FUNCTION_BLOCK FB_Device
VAR_INPUT
	inpAutomatic		: BOOL;
	inpSim				: BOOL := TRUE;
	
	cmdReset			: BOOL;
END_VAR
VAR_OUTPUT
END_VAR
VAR
END_VAR

PROPERTY ModeAutomatic : BOOL
GET
ModeAutomatic := inpAutomatic;
END_GET
END_PROPERTY

PROPERTY ModeManual : BOOL
GET
ModeManual := NOT inpAutomatic;
END_GET
END_PROPERTY

END_FUNCTION_BLOCK

(* stored: Version 1.1.0.1, ProductVersion 3.1.4024.4
   POU FB_Device: Id {df461c38-08f6-480c-a85c-0958733e653b}, SpecialFunc None
   Property ModeAutomatic: Id {15d02fd8-4ac5-4c34-9335-fe3f05621b5c}
   Get Get: Id {1cf7cdfc-1822-48eb-8dea-c7f604a7f1ff}
   Property ModeManual: Id {0b60a1fd-cf81-4142-a5ec-0c4baff3125e}
   Get Get: Id {d445e6da-51a0-4ea9-b1fd-0f122618dd5a} *)
